// TIA Portal V21 export
VAR_GLOBAL   // PLC tag table "Genericos"
   INSTR_01_STS_SEM_4mA AT %M5520.0 : Bool;
   INSTR_01_STS_LEITURA_ALTA AT %M5520.1 : Bool;
   INSTR_01_STS_LEITURA_BAIXA AT %M5520.2 : Bool;
   INSTR_01_STS_LEITURA_MUITO_ALTA AT %M5520.3 : Bool;
   INSTR_01_STS_LEITURA_MUITO_BAIXA AT %M5520.4 : Bool;
   MOTOR_01_STS_MOTOR_DESANERADOR_MODO_LOCAL_1 AT %M5520.5 : Bool;
   MOTOR_01_STS_MOTOR_DESANERADOR_MODO_REMOTO_1 AT %M5520.6 : Bool;
   QA_01_CMD_RESET_REMOTA AT %M5520.7 : Bool;
   CCM_01_STS_PAINEL_OK AT %M5521.0 : Bool;
   INSTR_01_PV_MACRO_MEDIDOR_VAZAO_INSTANTANEA AT %MD5522 : Real;
   INSTR_01_TOTALIZACAO_MEDIDOR_VAZAO AT %M5521.2 : Bool;
END_VAR
